TYPE ST_AutoMode_FeedInToWareHouseBox :
STRUCT
	Command 		: ST_FeedInToWareHouse_Ctrl;
	Status 			: ST_FeedInToWareHouse_Status;
	Info 			: ST_FeedInToWareHouseBox_Info;
	AClampMoveDone	: BOOL;
	BClampMoveDone	: BOOL;
END_STRUCT
END_TYPE

(* stored: Version 1.1.0.1, ProductVersion 3.1.4024.13
   DUT ST_AutoMode_FeedInToWareHouseBox: Id {a1b2c3d4-6666-4aaa-b666-666666666603} *)
